(* PLC project servo, Dassault Systèmes ControlBuild 2024x *)
(* stored: creationDateTime 2023-10-04T11:03:58-01:00 *)

(* This module assembles the different control/position/velocity parts *)
PROGRAM motion_control.servo
  VAR_IN_OUT
    status : INT := 0;
    errorFlag : INT := 0;
    ActualPositionAx1 : REAL := 0.0;
    MoveVelDone1 : BOOL := false;
    ActualVelocity1 : REAL := 0.0;
    MoveAbsDone1 : BOOL := false;
  END_VAR
  VAR_INPUT
    HomeCmd : BOOL := false;
    MoveVelCmd : BOOL := false;
    MoveAbsCmd : BOOL := false;
    MoveVel1ManualCmd : BOOL := false;
    MoveVel2ManualCmd : BOOL := false;
    MoveAbs1ManualCmd : BOOL := false;
    MoveAbs2ManualCmd : BOOL := false;
    StopCmd : BOOL := false;
    MovePosition : REAL := 0.0;
    MoveSpeed : REAL := 100.0;
    MoveAcceleration : REAL := 100.0;
    MoveDeceleration : REAL := 100.0;
    offsetAxToMa : REAL := 0.0;
  END_VAR
  VAR_INPUT
    PLC_StatusReady : BOOL := true;
    PLC_StatusMoved : BOOL := false;
    PLC_StatusStand : BOOL := false;
    PLC_ActualPositionAx : REAL := 0.0;
    PLC_ActualPositionMa : REAL := 0.0;
    PLC_ActualVelocity : REAL := 0.0;
  END_VAR
  VAR_INPUT
    physicalPosInit : REAL := 0.0;
    MAX_SPEED : REAL(0.0..3.4e+38) := 30.0;
    MAX_ACCEL : REAL(0.0..3.4e+38) := 1500.0;
    MAX_DECEL : REAL(0.0..3.4e+38) := 1500.0;
    MODULO_LENGTH : REAL := 0.0;
  END_VAR
  VAR_OUTPUT
    StatusReady : BOOL := true;
    StatusMoved : BOOL := false;
    StatusStand : BOOL := false;
    ActualPositionAx : REAL := 0.0;
    ActualPositionMa : REAL := 0.0;
    ActualVelocity : REAL := 0.0;
    MaximumVelocity : REAL := 0.0;
    StatusPosIncrease : BOOL := false;
    StatusPosDecrease : BOOL := false;
    displayJauge : REAL := 0.0;
  END_VAR

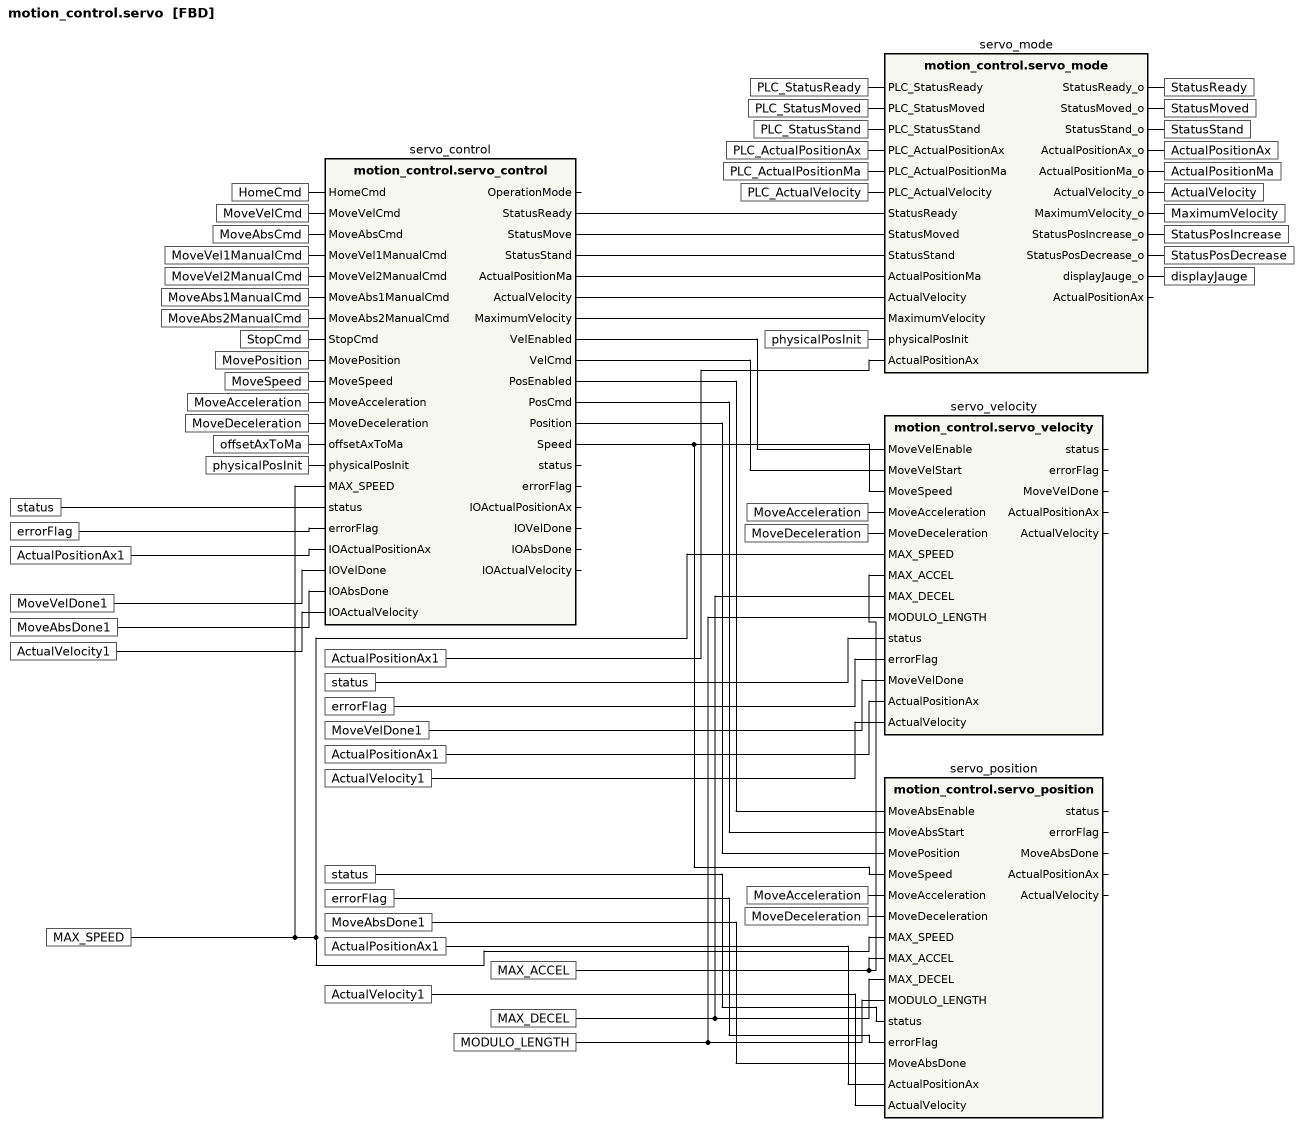
(* FBD diagram, written out as Structured Text *)
servo_control(HomeCmd := HomeCmd, MoveVelCmd := MoveVelCmd, MoveAbsCmd := MoveAbsCmd, MoveVel1ManualCmd := MoveVel1ManualCmd, MoveVel2ManualCmd := MoveVel2ManualCmd, MoveAbs1ManualCmd := MoveAbs1ManualCmd, MoveAbs2ManualCmd := MoveAbs2ManualCmd, StopCmd := StopCmd, MovePosition := MovePosition, MoveSpeed := MoveSpeed, MoveAcceleration := MoveAcceleration, MoveDeceleration := MoveDeceleration, offsetAxToMa := offsetAxToMa, physicalPosInit := physicalPosInit, MAX_SPEED := MAX_SPEED, status := status, errorFlag := errorFlag, IOActualPositionAx := ActualPositionAx1, IOVelDone := MoveVelDone1, IOAbsDone := MoveAbsDone1, IOActualVelocity := ActualVelocity1);
servo_mode(PLC_StatusReady := PLC_StatusReady, PLC_StatusMoved := PLC_StatusMoved, PLC_StatusStand := PLC_StatusStand, PLC_ActualPositionAx := PLC_ActualPositionAx, PLC_ActualPositionMa := PLC_ActualPositionMa, PLC_ActualVelocity := PLC_ActualVelocity, StatusReady := servo_control.StatusReady, StatusMoved := servo_control.StatusMove, StatusStand := servo_control.StatusStand, ActualPositionMa := servo_control.ActualPositionMa, ActualVelocity := servo_control.ActualVelocity, MaximumVelocity := servo_control.MaximumVelocity, physicalPosInit := physicalPosInit, ActualPositionAx := ActualPositionAx1);
StatusReady := servo_mode.StatusReady_o;
StatusMoved := servo_mode.StatusMoved_o;
StatusStand := servo_mode.StatusStand_o;
ActualPositionAx := servo_mode.ActualPositionAx_o;
ActualPositionMa := servo_mode.ActualPositionMa_o;
ActualVelocity := servo_mode.ActualVelocity_o;
MaximumVelocity := servo_mode.MaximumVelocity_o;
StatusPosIncrease := servo_mode.StatusPosIncrease_o;
StatusPosDecrease := servo_mode.StatusPosDecrease_o;
displayJauge := servo_mode.displayJauge_o;
servo_velocity(MoveVelEnable := servo_control.VelEnabled, MoveVelStart := servo_control.VelCmd, MoveSpeed := servo_control.Speed, MoveAcceleration := MoveAcceleration, MoveDeceleration := MoveDeceleration, MAX_SPEED := MAX_SPEED, MAX_ACCEL := MAX_ACCEL, MAX_DECEL := MAX_DECEL, MODULO_LENGTH := MODULO_LENGTH, status := status, errorFlag := errorFlag, MoveVelDone := MoveVelDone1, ActualPositionAx := ActualPositionAx1, ActualVelocity := ActualVelocity1);
servo_position(MoveAbsEnable := servo_control.PosEnabled, MoveAbsStart := servo_control.PosCmd, MovePosition := servo_control.Position, MoveSpeed := servo_control.Speed, MoveAcceleration := MoveAcceleration, MoveDeceleration := MoveDeceleration, MAX_SPEED := MAX_SPEED, MAX_ACCEL := MAX_ACCEL, MAX_DECEL := MAX_DECEL, MODULO_LENGTH := MODULO_LENGTH, status := status, errorFlag := errorFlag, MoveAbsDone := MoveAbsDone1, ActualPositionAx := ActualPositionAx1, ActualVelocity := ActualVelocity1);
END_PROGRAM
